TYPE LogArrayHandlePointers :
STRUCT
	writePointer : UINT := 0;
	readPointer : UINT := 0;
	numOfMembers : UINT := 0;
	isBusy : BOOL := FALSE; (*If writing to array is busy now*)
END_STRUCT
END_TYPE

(* stored: Version 1.1.0.1, ProductVersion 3.1.4024.3
   DUT LogArrayHandlePointers: Id {0bdfd265-aff5-0db6-101c-b32a3e642899} *)
